(* PLC project Proyecto, Unknown Unnamed 1 *)
(* stored: creationDateTime 2025-03-16T15:34:21, modificationDateTime 2025-04-12T20:39:13 *)

TYPE FSM1_TSTATUS : (FSM1_ESPERA, FSM1_ARRANCANDO_BANDAS, FSM1_ESPERANDO_CLASIFICACION, FSM1_ESPERANDO_DETECCION_PIEZA, FSM1_CLAMPEANDO, FSM1_RECOGIENDO_PIEZA_SUCCIONADOR1, FSM1_RECOGIENDO_CAJA_SUCCIONADOR2);
END_TYPE

TYPE FSM1_TRANSITIONS : (FSM1_INICIAR, FSM1_DESHABILITADO, FSM1_CLASIFICAR_CAJAS_COLOR, FSM1_DETECTAR_PIEZA_EMPUJAR, FSM1_CLAMPEAR, FSM1_RECOGER_PIEZA_SUCCIONADOR1, FSM1_RECOGER_CAJA_SUCCIONADOR2);
END_TYPE

TYPE FSM2_TSTATUS : (FSM2_NULLL, FSM2_VALIDANDO_TRANSACCION, FSM2_INICIANDO_SECUENCIA);
END_TYPE

TYPE FSM2_TTRANSITIONS : (FSM2_DESHABILITADO, FSM2_INICIAR_SECUENCIA, FSM2_DETECTAR_PALLET);
END_TYPE

FUNCTION_BLOCK FSM1_Petri
  VAR_EXTERNAL
    FSM1_CurrentTransition : FSM1_TRANSITIONS;
    FSM1_CurrentStatus : FSM1_TSTATUS;
  END_VAR

            (*Red FSM1_Petri*)
IF FSM1_CurrentTransition = FSM1_INICIAR 
  THEN
    FSM1_CurrentStatus:=FSM1_ARRANCANDO_BANDAS;
END_IF;

IF FSM1_CurrentTransition = FSM1_CLASIFICAR_CAJAS_COLOR 
  THEN
    FSM1_CurrentStatus:=FSM1_ESPERANDO_CLASIFICACION;
END_IF;

IF FSM1_CurrentTransition = FSM1_DETECTAR_PIEZA_EMPUJAR
    THEN
      FSM1_CurrentStatus:=FSM1_ESPERANDO_DETECCION_PIEZA;
END_IF;

IF FSM1_CurrentTransition = FSM1_CLAMPEAR
    THEN
      FSM1_CurrentStatus:=FSM1_CLAMPEANDO;
END_IF;

IF FSM1_CurrentTransition = FSM1_RECOGER_PIEZA_SUCCIONADOR1
  THEN
      FSM1_CurrentStatus:=FSM1_RECOGIENDO_PIEZA_SUCCIONADOR1;
END_IF;

IF FSM1_CurrentTransition = FSM1_RECOGER_CAJA_SUCCIONADOR2

  THEN

      FSM1_CurrentStatus:=FSM1_RECOGIENDO_CAJA_SUCCIONADOR2;

END_IF;
          
END_FUNCTION_BLOCK

FUNCTION_BLOCK FSM1_Triggers
  VAR_EXTERNAL
    FSM1_CurrentStatus : FSM1_TSTATUS;
    FSM1_CurrentTransition : FSM1_TRANSITIONS;
  END_VAR
  VAR
    FSM1_FTrigStop : F_TRIG;
  END_VAR
  VAR_EXTERNAL
    FSM1_RCSorting1 : BOOL;
    FSM1_RCSorting2 : BOOL;
    FSM1_RCSorting3 : BOOL;
    FSM1_RCSorting4 : BOOL;
    FSM1_RCSorting5 : BOOL;
    FSM1_RCSorting6 : BOOL;
    FSM1_RCSorting7 : BOOL;
    FSM1_RCSorting8 : BOOL;
    FSM1_RCSorting9 : BOOL;
    FSM1_BtnStop : BOOL;
    FSM1_BtnStart : BOOL;
    FSM1_SensorVision1 : INT;
  END_VAR
  VAR
    SensorVision1Value : INT;
  END_VAR
  VAR_EXTERNAL
    FSM1_SensorPusher1 : BOOL;
    FSM1_SensorPusher2 : BOOL;
    FSM1_PusherSorting1 : BOOL;
    FSM1_PusherSorting2 : BOOL;
  END_VAR
  VAR
    TP_Pusher1 : TP;
    TP_Pusher2 : TP;
  END_VAR
  VAR_EXTERNAL
    FSM1_RCGreen : BOOL;
    FSM1_RCBlue : BOOL;
  END_VAR
  VAR
    FTRIG_Pusher1 : F_TRIG;
    FTRIG_Pusher2 : F_TRIG;
    FTRIG_SensorClampBlue : F_TRIG;
  END_VAR
  VAR_EXTERNAL
    FSM1_SensorClampBlue : BOOL;
    FSM1_SensorClampGreen : BOOL;
    FSM1_OutClampBlue : BOOL;
    FSM1_OutClampGreen : BOOL;
  END_VAR
  VAR
    TP_ClampBlue : TP;
    FTRIG_ClampBlue : F_TRIG;
  END_VAR
  VAR_EXTERNAL
    BASE_BLUE : INT;
    LID_BLUE : INT;
    LID_GREEN : INT;
    BASE_GREEN : INT;
  END_VAR
  VAR
    FTRIG_SensorClampGreen : F_TRIG;
    TP_ClampGreen : TP;
    FTRIG_ClampGreen : F_TRIG;
  END_VAR
  VAR_EXTERNAL
    FSM1_Sucker1X : INT;
    FSM1_Sucker1Y : INT;
    FSM1_Sucker1Z : INT;
  END_VAR
  VAR
    TON_Sucker1 : TON;
    FSM_Sucker1 : INT := 0;
  END_VAR
  VAR_EXTERNAL
    FSM1_OutSucker1Grab : BOOL;
  END_VAR

            FSM1_FTrigStop(

     CLK := FSM1_BtnStop
);

IF FSM1_FTrigStop.Q THEN
  FSM1_CurrentTransition:=FSM1_DESHABILITADO;
  FSM1_CurrentStatus:= FSM1_ESPERA;
  SensorVision1Value:=0;
  FSM1_RCSorting1:=FALSE;
  FSM1_RCSorting2:=FALSE;
  FSM1_RCSorting3:=FALSE;
  FSM1_RCSorting4:=FALSE;
  FSM1_RCSorting5:=FALSE;
  FSM1_RCSorting6:=FALSE;
  FSM1_RCSorting7:=FALSE;
  FSM1_RCSorting8:=FALSE;
  FSM1_RCSorting9:=FALSE;
  FSM1_RCGreen:=FALSE;
  FSM1_RCBlue:=FALSE;
  FSM1_OutSucker1Grab := FALSE;

  FSM1_Sucker1Z := 0;
  FSM1_Sucker1Y := 0;
  FSM1_Sucker1X := 0;
END_IF;

IF FSM1_CurrentStatus = FSM1_ESPERA
  THEN
  IF FSM1_BtnStart
    THEN
      FSM1_CurrentTransition:= FSM1_INICIAR;
  END_IF;
END_IF;

IF FSM1_CurrentStatus = FSM1_ARRANCANDO_BANDAS
  THEN
      FSM1_RCSorting1:=TRUE;
      FSM1_RCSorting2:=TRUE;
      FSM1_RCSorting3:=TRUE;
      FSM1_RCSorting4:=TRUE;
      FSM1_RCSorting5:=TRUE;
      FSM1_RCSorting6:=TRUE;
      FSM1_RCSorting7:=TRUE;
      FSM1_RCSorting8:=TRUE;
      FSM1_RCSorting9:=TRUE;
      FSM1_RCGreen:=TRUE;
      FSM1_RCBlue:=TRUE;
      SensorVision1Value:=0;
      FSM1_CurrentTransition:=FSM1_CLASIFICAR_CAJAS_COLOR;
END_IF;

IF FSM1_CurrentStatus = FSM1_ESPERANDO_CLASIFICACION 
  THEN
    IF FSM1_SensorVision1 > 0 THEN
      SensorVision1Value:= FSM1_SensorVision1;    
      FSM1_CurrentTransition := FSM1_DETECTAR_PIEZA_EMPUJAR;
    END_IF;
END_IF;

IF FSM1_CurrentStatus =FSM1_ESPERANDO_DETECCION_PIEZA 
    THEN
      IF  SensorVision1Value = LID_GREEN OR 
          SensorVision1Value = BASE_GREEN
      THEN
        TP_Pusher1(
         IN := FSM1_SensorPusher1,
         PT := T#2s,
         Q => FSM1_PusherSorting1
        );
        FTRIG_Pusher1(
            CLK := TP_Pusher1.Q
          );
        IF FTRIG_Pusher1.Q 

          THEN

           FSM1_CurrentTransition := FSM1_CLAMPEAR;

        END_IF;
      END_IF;
      
      IF  SensorVision1Value = LID_BLUE OR 
          SensorVision1Value = BASE_BLUE
        THEN
          TP_Pusher2(
           IN := FSM1_SensorPusher2,
           PT := T#2s,
           Q => FSM1_PusherSorting2
          );
          FTRIG_Pusher2(
            CLK:= TP_Pusher2.Q
          );
          IF FTRIG_Pusher2.Q 
            THEN
            FSM1_CurrentTransition := FSM1_CLAMPEAR;
          END_IF;
      END_IF;
      
END_IF;


IF FSM1_CurrentStatus = FSM1_CLAMPEANDO 
  THEN
    IF  SensorVision1Value = LID_BLUE OR 

          SensorVision1Value = BASE_BLUE

      THEN
      (*Detectar cuando la pieza ha pasado por completo el sensor*)

      FTRIG_SensorClampBlue(

         CLK := FSM1_SensorClampBlue

      );

      TP_ClampBlue(

         IN := FTRIG_SensorClampBlue.Q ,

         PT := T#1s,

         Q => FSM1_OutClampBlue

       );

      FTRIG_ClampBlue(

        CLK := TP_ClampBlue.Q

       );

      IF FTRIG_ClampBlue.Q THEN

        FSM1_CurrentTransition:=FSM1_RECOGER_PIEZA_SUCCIONADOR1;

      END_IF;
  END_IF;
  
  IF  SensorVision1Value = LID_GREEN OR 

          SensorVision1Value = BASE_GREEN

    THEN
      (*Detectar cuando la pieza ha pasado por completo el sensor*)

      FTRIG_SensorClampGreen(

         CLK := FSM1_SensorClampGreen

      );

      TP_ClampGreen(

         IN := FTRIG_SensorClampGreen.Q ,

         PT := T#1s,

         Q => FSM1_OutClampGreen

       );

      FTRIG_ClampGreen(

        CLK := TP_ClampGreen.Q

       );

      IF FTRIG_ClampGreen.Q THEN

        FSM1_CurrentTransition:=FSM1_RECOGER_PIEZA_SUCCIONADOR1;

      END_IF;
  END_IF;
END_IF;

IF FSM1_CurrentStatus = FSM1_RECOGIENDO_PIEZA_SUCCIONADOR1
  THEN
  IF  SensorVision1Value = LID_BLUE OR 

          SensorVision1Value = BASE_BLUE

    THEN
    CASE FSM_Sucker1 OF

      0:(*Primer paso*) 

        FSM1_Sucker1Z := 8;

        TON_Sucker1(IN := TRUE, PT := T#2s); 

        IF TON_Sucker1.Q THEN

          TON_Sucker1(IN := FALSE); 

          FSM_Sucker1:= 1;

        END_IF;



      1:(*Segundo paso*)

        FSM1_Sucker1X := 1;

        TON_Sucker1(IN := TRUE, PT := T#2s); 

        IF TON_Sucker1.Q THEN

          TON_Sucker1(IN := FALSE);

          FSM_Sucker1:= 2;

        END_IF;



      2: (*Activar succión*)

        FSM1_OutSucker1Grab := TRUE;

        FSM1_Sucker1Z := 0;

        FSM_Sucker1:= 3;
        

      3: (*Fin o esperar nueva orden*)

        FSM1_CurrentTransition:=FSM1_RECOGER_CAJA_SUCCIONADOR2;

    END_CASE;
  END_IF;
  
    IF  SensorVision1Value = LID_GREEN OR 

          SensorVision1Value = BASE_GREEN

      THEN
        CASE FSM_Sucker1 OF

        0:(*Primer paso*) 

          FSM1_Sucker1X := 8;

          TON_Sucker1(IN := TRUE, PT := T#2s); 

          IF TON_Sucker1.Q THEN

            TON_Sucker1(IN := FALSE); 

            FSM_Sucker1:= 1;

          END_IF;



        1:(*Segundo paso*)

          FSM1_Sucker1Z := 8;

          TON_Sucker1(IN := TRUE, PT := T#2s); 

          IF TON_Sucker1.Q THEN

            TON_Sucker1(IN := FALSE);

            FSM_Sucker1:= 2;

          END_IF;



        2: (*Activar succión*)

          FSM1_OutSucker1Grab := TRUE;

          FSM1_Sucker1Z := 0;

          FSM_Sucker1:= 3;

          

        3: (*Fin o esperar nueva orden*)

          FSM1_CurrentTransition:=FSM1_RECOGER_CAJA_SUCCIONADOR2;

      END_CASE;
    END_IF;

      
END_IF;
      
      
          
            

          
END_FUNCTION_BLOCK

PROGRAM main
  VAR
    FSM1_Petri0 : FSM1_Petri;
    FSM1_Triggers0 : FSM1_Triggers;
  END_VAR

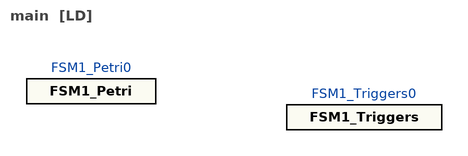
(* LD diagram, written out as Structured Text *)
FSM1_Petri0();
FSM1_Triggers0();
END_PROGRAM

CONFIGURATION Config0
  RESOURCE Res0 ON PLC
    VAR_GLOBAL
      FSM1_CurrentStatus : FSM1_TSTATUS := FSM1_ESPERA;
      FSM1_CurrentTransition : FSM1_TRANSITIONS := FSM1_DESHABILITADO;
      FSM2_CurrentTransition : FSM2_TTRANSITIONS := FSM2_DESHABILITADO;
      FSM2_CurrentStatus : FSM2_TSTATUS := FSM2_VALIDANDO_TRANSACCION;
      FSM1_BtnStart AT %IX100.0 : BOOL := FALSE;
      FSM1_BtnStop AT %IX100.1 : BOOL := TRUE;
      FSM1_SensorPusher1 AT %IX100.2 : BOOL := TRUE;
      FSM1_SensorPusher2 AT %IX100.3 : BOOL := TRUE;
      FSM1_SensorClampBlue AT %IX100.4 : BOOL := TRUE;
      FSM1_SensorClampGreen AT %IX100.5 : BOOL := TRUE;
      FSM1_RCSorting1 AT %QX100.0 : BOOL := FALSE;
      FSM1_RCSorting2 AT %QX100.1 : BOOL := FALSE;
      FSM1_RCSorting3 AT %QX100.2 : BOOL := FALSE;
      FSM1_RCSorting4 AT %QX100.3 : BOOL := FALSE;
      FSM1_RCSorting5 AT %QX100.4 : BOOL := FALSE;
      FSM1_RCSorting6 AT %QX100.5 : BOOL := FALSE;
      FSM1_RCSorting7 AT %QX100.6 : BOOL := FALSE;
      FSM1_RCSorting8 AT %QX100.7 : BOOL := FALSE;
      FSM1_RCSorting9 AT %QX101.0 : BOOL := FALSE;
      FSM1_PusherSorting1 AT %QX101.1 : BOOL := FALSE;
      FSM1_PusherSorting2 AT %QX101.2 : BOOL := FALSE;
      FSM1_RcGreen AT %QX101.3 : BOOL := FALSE;
      FSM1_RcBlue AT %QX101.4 : BOOL := FALSE;
      FSM1_OutClampBlue AT %QX101.5 : BOOL := FALSE;
      FSM1_OutClampGreen AT %QX101.6 : BOOL := FALSE;
      FSM1_OutSucker1Grab AT %QX101.7 : BOOL := FALSE;
      FSM1_SensorVision1 AT %IW100 : INT := 0;
      FSM1_SensorVision2 AT %IW101 : INT := 0;
      FSM1_Sucker1X AT %QW100 : INT := 0;
      FSM1_Sucker1Y AT %QW101 : INT := 0;
      FSM1_Sucker1Z AT %QW102 : INT := 0;
      BASE_BLUE : INT := 3;
      BASE_GREEN : INT := 6;
      LID_GREEN : INT := 5;
      LID_BLUE : INT := 2;
    END_VAR
    TASK task0(INTERVAL := T#20ms, PRIORITY := 0);
    PROGRAM instance0 WITH task0 : main;
  END_RESOURCE
END_CONFIGURATION
